FUNCTION Chek_Buffer_Layout : Buffer_Layout_Error
VAR_INPUT
	Layout : REFERENCE TO Buffer_Layout;
END_VAR

VAR
	Current_Buffer_Size : USINT := 0;
	i : UINT;
	LowerBoud : USINT;
	UpperBound : USINT;
END_VAR

// calculate buffer size
// Bool array
IF Layout.Enabel_Bool_Array THEN 
	Current_Buffer_Size := Layout.Bool_Amount * 1; 
END_IF;
// SInt array
IF Layout.Enabel_SInt_Array THEN 
	Current_Buffer_Size := Current_Buffer_Size + (Layout.SInt_Amount * 8); 
END_IF;
// USInt array
IF Layout.Enabel_USInt_Array THEN 
	Current_Buffer_Size := Current_Buffer_Size + (Layout.USInt_Amount * 8);
END_IF;
// Int array
IF Layout.Enabel_Int_Array THEN
	Current_Buffer_Size := Current_Buffer_Size + (Layout.Int_Amount * 16);
END_IF;
// UInt array
IF Layout.Enabel_UInt_Array THEN
	Current_Buffer_Size := Current_Buffer_Size + (Layout.UInt_Amount * 16);
END_IF;
// DInt array
IF Layout.Enabel_DInt_Array THEN
	Current_Buffer_Size := Current_Buffer_Size + (Layout.DInt_Amount * 32);
END_IF;
// UDInt array
IF Layout.Enabel_UDInt_Array THEN
	Current_Buffer_Size := Current_Buffer_Size + (Layout.UDInt_Amount * 32);
END_IF;
// Real array
IF Layout.Enabel_Real_Array THEN
	Current_Buffer_Size := Current_Buffer_Size + (Layout.Real_Amount * 32);
END_IF;
// String array
IF Layout.Enabel_String_Array THEN
	FOR i:=0 TO 3 BY 1 DO
		Current_Buffer_Size := Current_Buffer_Size + (Layout.String_Amount * Layout.String_Lengts[i]);
	END_FOR
END_IF;

IF Layout.Buffer_Size > Current_Buffer_Size THEN
	Chek_Buffer_Layout := Chek_Buffer_Layout OR Buffer_Layout_Error.Overflow;
END_IF


// overlay chek
// Bool array
LowerBoud := Layout.Bool_Array_Offset;
UpperBound := Layout.Bool_Array_Offset * Layout.Bool_Amount;
IF Overlap_Chek(Layout:= Layout, Array_Type:= Layout_Array_Types.Bool_Type, LowerBound_Target:= LowerBoud, UpperBound_Target:= UpperBound) THEN
	Chek_Buffer_Layout := Chek_Buffer_Layout OR Buffer_Layout_Error.Overlap;
END_IF

// SInt array
LowerBoud := Layout.SInt_Array_Offset;
UpperBound := Layout.SInt_Array_Offset * Layout.SInt_Amount;
IF Overlap_Chek(Layout:= Layout, Array_Type:= Layout_Array_Types.SInt_Type, LowerBound_Target:= LowerBoud, UpperBound_Target:= UpperBound) THEN
	Chek_Buffer_Layout := Chek_Buffer_Layout OR Buffer_Layout_Error.Overlap;
END_IF

// USInt array
LowerBoud := Layout.USInt_Array_Offset;
UpperBound := Layout.USInt_Array_Offset * Layout.USInt_Amount;
IF Overlap_Chek(Layout:= Layout, Array_Type:= Layout_Array_Types.USInt_Type, LowerBound_Target:= LowerBoud, UpperBound_Target:= UpperBound) THEN
	Chek_Buffer_Layout := Chek_Buffer_Layout OR Buffer_Layout_Error.Overlap;
END_IF

// Int array
LowerBoud := Layout.Int_Array_Offset;
UpperBound := Layout.Int_Array_Offset * Layout.Int_Amount;
IF Overlap_Chek(Layout:= Layout, Array_Type:= Layout_Array_Types.Int_Type, LowerBound_Target:= LowerBoud, UpperBound_Target:= UpperBound) THEN
	;
END_IF

// UInt array
LowerBoud := Layout.UInt_Array_Offset;
UpperBound := Layout.UInt_Array_Offset * Layout.UInt_Amount;
IF Overlap_Chek(Layout:= Layout, Array_Type:= Layout_Array_Types.UInt_Type, LowerBound_Target:= LowerBoud, UpperBound_Target:= UpperBound) THEN
	Chek_Buffer_Layout := Chek_Buffer_Layout OR Buffer_Layout_Error.Overlap;
END_IF

// DInt array
LowerBoud := Layout.DInt_Array_Offset;
UpperBound := Layout.DInt_Array_Offset * Layout.DInt_Amount;
IF Overlap_Chek(Layout:= Layout, Array_Type:= Layout_Array_Types.DInt_Type, LowerBound_Target:= LowerBoud, UpperBound_Target:= UpperBound) THEN
	Chek_Buffer_Layout := Chek_Buffer_Layout OR Buffer_Layout_Error.Overlap;
END_IF

// UDInt array
LowerBoud := Layout.UDInt_Array_Offset;
UpperBound := Layout.UDInt_Array_Offset * Layout.UDInt_Amount;
IF Overlap_Chek(Layout:= Layout, Array_Type:= Layout_Array_Types.UDInt_Type, LowerBound_Target:= LowerBoud, UpperBound_Target:= UpperBound) THEN
	Chek_Buffer_Layout := Chek_Buffer_Layout OR Buffer_Layout_Error.Overlap;
END_IF

// Real array
LowerBoud := Layout.Real_Array_Offset;
UpperBound := Layout.Real_Array_Offset * Layout.Real_Amount;
IF Overlap_Chek(Layout:= Layout, Array_Type:= Layout_Array_Types.Real_Type, LowerBound_Target:= LowerBoud, UpperBound_Target:= UpperBound) THEN
	Chek_Buffer_Layout := Chek_Buffer_Layout OR Buffer_Layout_Error.Overlap;
END_IF

// String array
LowerBoud := Layout.String_Array_Offset;
UpperBound := 0;
FOR i:=0 TO Layout.String_Amount BY 1 DO
	UpperBound := UpperBound + Layout.String_Lengts[i];
END_FOR
IF Overlap_Chek(Layout:= Layout, Array_Type:= Layout_Array_Types.String_Type, LowerBound_Target:= LowerBoud, UpperBound_Target:= UpperBound) THEN
	Chek_Buffer_Layout := Chek_Buffer_Layout OR Buffer_Layout_Error.Overlap;
END_IF

END_FUNCTION

(* stored: Version 1.1.0.1, ProductVersion 3.1.4024.10
   POU Chek_Buffer_Layout: Id {2be24f20-7608-4a8e-a150-78d6070c33de}, SpecialFunc None *)
